TYPE PLCToHMIOperatingMode :
STRUCT
	CurrentOperatingMode	:	OperatingMode;	
END_STRUCT
END_TYPE

(* stored: Version 1.1.0.1
   DUT PLCToHMIOperatingMode: Id {95cbae51-f4ba-43cf-905a-89be056966bd} *)
